Fanuc TP program (LS listing): WALL.LS

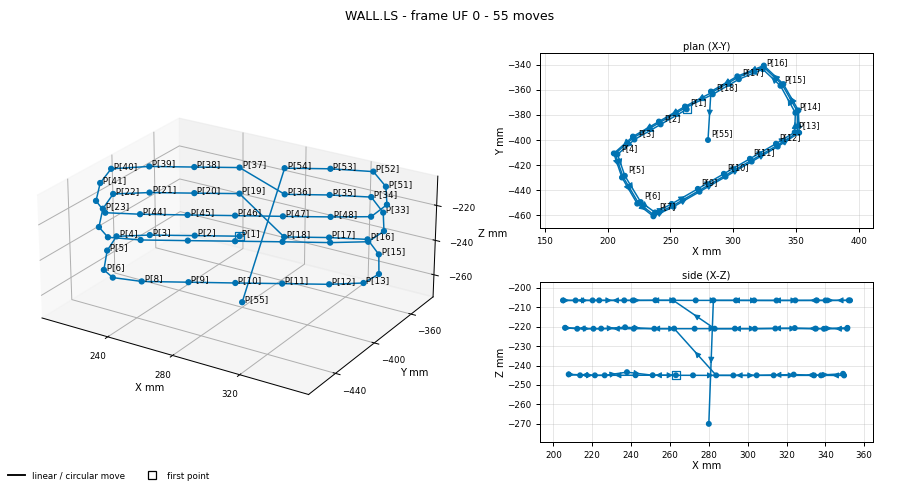
[picture p0: tool path of WALL.LS in frame UF 0, 55 of 55 moves have a stored position in this frame; points joined in program order, loops and branches not executed]
/PROG  WALL.LS
/ATTR
OWNER       = MNEDITOR;
COMMENT     = "";
PROG_SIZE   = 636;
CREATE      = DATE 23-01-07  TIME 11:59:14;
MODIFIED    = DATE 23-01-07  TIME 12:02:18;
FILE_NAME   = ;
VERSION     = 0;
LINE_COUNT  = 4;
MEMORY_SIZE = 992;
PROTECT     = READ_WRITE;
TCD:  STACK_SIZE	= 0,
      TASK_PRIORITY	= 50,
      TIME_SLICE	= 0,
      BUSY_LAMP_OFF	= 0,
      ABORT_REQUEST	= 0,
      PAUSE_REQUEST	= 0;
DEFAULT_GROUP	= 1,*,*,*,*;
CONTROL_CODE	= 00000000 00000000;
/MN
   1:J P[1] 100% FINE    ;
   2:L P[2] 100mm/sec CNT0    ;
   3:L P[3] 100mm/sec CNT0    ;
   4:L P[4] 100mm/sec CNT0    ;
   5:L P[5] 100mm/sec CNT0    ;
   6:L P[6] 100mm/sec CNT0    ;
   7:L P[7] 100mm/sec CNT0    ;
   8:L P[8] 100mm/sec CNT0    ;
   9:L P[9] 100mm/sec CNT0    ;
   10:L P[10] 100mm/sec CNT0    ;
   11:L P[11] 100mm/sec CNT0    ;
   12:L P[12] 100mm/sec CNT0    ;
   13:L P[13] 100mm/sec CNT0    ;
   14:L P[14] 100mm/sec CNT0    ;
   15:L P[15] 100mm/sec CNT0    ;
   16:L P[16] 100mm/sec CNT0    ;
   17:L P[17] 100mm/sec CNT0    ;
   18:L P[18] 100mm/sec CNT0    ;
   19:L P[19] 100mm/sec CNT0    ;
   20:L P[20] 100mm/sec CNT0    ;
   21:L P[21] 100mm/sec CNT0    ;
   22:L P[22] 100mm/sec CNT0    ;
   23:L P[23] 100mm/sec CNT0    ;
   24:L P[24] 100mm/sec CNT0    ;
   25:L P[25] 100mm/sec CNT0    ;
   26:L P[26] 100mm/sec CNT0    ;
   27:L P[27] 100mm/sec CNT0    ;
   28:L P[28] 100mm/sec CNT0    ;
   29:L P[29] 100mm/sec CNT0    ;
   30:L P[30] 100mm/sec CNT0    ;
   31:L P[31] 100mm/sec CNT0    ;
   32:L P[32] 100mm/sec CNT0    ;
   33:L P[33] 100mm/sec CNT0    ;
   34:L P[34] 100mm/sec CNT0    ;
   35:L P[35] 100mm/sec CNT0    ;
   36:L P[36] 100mm/sec CNT0    ;
   37:L P[37] 100mm/sec CNT0    ;
   38:L P[38] 100mm/sec CNT0    ;
   39:L P[39] 100mm/sec CNT0    ;
   40:L P[40] 100mm/sec CNT0    ;
   41:L P[41] 100mm/sec CNT0    ;
   42:L P[42] 100mm/sec CNT0    ;
   43:L P[43] 100mm/sec CNT0    ;
   44:L P[44] 100mm/sec CNT0    ;
   45:L P[45] 100mm/sec CNT0    ;
   46:L P[46] 100mm/sec CNT0    ;
   47:L P[47] 100mm/sec CNT0    ;
   48:L P[48] 100mm/sec CNT0    ;
   49:L P[49] 100mm/sec CNT0    ;
   50:L P[50] 100mm/sec CNT0    ;
   51:L P[51] 100mm/sec CNT0    ;
   52:L P[52] 100mm/sec CNT0    ;
   53:L P[53] 100mm/sec CNT0    ;
   54:L P[54] 100mm/sec CNT0    ;
   55:L P[55] 100mm/sec CNT0    ;
/POS
P[1]{
   GP1:
	UF : 0, UT : 6,		CONFIG : 'N U T, 0, 0, 0',
	X =  263.064  mm,	Y =   -375.561  mm,	Z =   -244.966  mm,
	W =  90.000 deg,	P =   0.000 deg,	R =   90.000 deg
};
P[2]{
   GP1:
	UF : 0, UT : 6,		CONFIG : 'N U T, 0, 0, 0',
	X =  242.275  mm,	Y =   -387.566  mm,	Z =   -244.990  mm,
	W =  90.000 deg,	P =   0.000 deg,	R =   90.000 deg
};
P[3]{
   GP1:
	UF : 0, UT : 6,		CONFIG : 'N U T, 0, 0, 0',
	X =  221.367  mm,	Y =   -399.643  mm,	Z =   -245.032  mm,
	W =  90.000 deg,	P =   0.000 deg,	R =   90.000 deg
};
P[4]{
   GP1:
	UF : 0, UT : 6,		CONFIG : 'N U T, 0, 0, 0',
	X =  207.874  mm,	Y =   -411.456  mm,	Z =   -244.528  mm,
	W =  90.000 deg,	P =   0.000 deg,	R =   90.000 deg
};
P[5]{
   GP1:
	UF : 0, UT : 6,		CONFIG : 'N U T, 0, 0, 0',
	X =  213.737  mm,	Y =   -428.487  mm,	Z =   -245.003  mm,
	W =  90.000 deg,	P =   0.000 deg,	R =   90.000 deg
};
P[6]{
   GP1:
	UF : 0, UT : 6,		CONFIG : 'N U T, 0, 0, 0',
	X =  226.401  mm,	Y =   -449.442  mm,	Z =   -245.036  mm,
	W =  90.000 deg,	P =   0.000 deg,	R =   90.000 deg
};
P[7]{
   GP1:
	UF : 0, UT : 6,		CONFIG : 'N U T, 0, 0, 0',
	X =  237.864  mm,	Y =   -457.694  mm,	Z =   -243.394  mm,
	W =  90.000 deg,	P =   0.000 deg,	R =   90.000 deg
};
P[8]{
   GP1:
	UF : 0, UT : 6,		CONFIG : 'N U T, 0, 0, 0',
	X =  251.098  mm,	Y =   -450.903  mm,	Z =   -244.977  mm,
	W =  90.000 deg,	P =   0.000 deg,	R =   90.000 deg
};
P[9]{
   GP1:
	UF : 0, UT : 6,		CONFIG : 'N U T, 0, 0, 0',
	X =  271.875  mm,	Y =   -438.904  mm,	Z =   -245.024  mm,
	W =  90.000 deg,	P =   0.000 deg,	R =   90.000 deg
};
P[10]{
   GP1:
	UF : 0, UT : 6,		CONFIG : 'N U T, 0, 0, 0',
	X =  292.641  mm,	Y =   -426.910  mm,	Z =   -245.078  mm,
	W =  90.000 deg,	P =   0.000 deg,	R =   90.000 deg
};
P[11]{
   GP1:
	UF : 0, UT : 6,		CONFIG : 'N U T, 0, 0, 0',
	X =  313.392  mm,	Y =   -414.931  mm,	Z =   -245.046  mm,
	W =  90.000 deg,	P =   0.000 deg,	R =   90.000 deg
};
P[12]{
   GP1:
	UF : 0, UT : 6,		CONFIG : 'N U T, 0, 0, 0',
	X =  334.179  mm,	Y =   -402.928  mm,	Z =   -245.053  mm,
	W =  90.000 deg,	P =   0.000 deg,	R =   90.000 deg
};
P[13]{
   GP1:
	UF : 0, UT : 6,		CONFIG : 'N U T, 0, 0, 0',
	X =  349.100  mm,	Y =   -393.829  mm,	Z =   -244.223  mm,
	W =  90.000 deg,	P =   0.000 deg,	R =   90.000 deg
};
P[14]{
   GP1:
	UF : 0, UT : 6,		CONFIG : 'N U T, 0, 0, 0',
	X =  349.628  mm,	Y =   -378.344  mm,	Z =   -245.091  mm,
	W =  90.000 deg,	P =   0.000 deg,	R =   90.000 deg
};
P[15]{
   GP1:
	UF : 0, UT : 6,		CONFIG : 'N U T, 0, 0, 0',
	X =  337.749  mm,	Y =   -356.772  mm,	Z =   -245.043  mm,
	W =  90.000 deg,	P =   0.000 deg,	R =   90.000 deg
};
P[16]{
   GP1:
	UF : 0, UT : 6,		CONFIG : 'N U T, 0, 0, 0',
	X =  323.686  mm,	Y =   -343.563  mm,	Z =   -244.638  mm,
	W =  90.000 deg,	P =   0.000 deg,	R =   90.000 deg
};
P[17]{
   GP1:
	UF : 0, UT : 6,		CONFIG : 'N U T, 0, 0, 0',
	X =  304.635  mm,	Y =   -351.562  mm,	Z =   -245.020  mm,
	W =  90.000 deg,	P =   0.000 deg,	R =   90.000 deg
};
P[18]{
   GP1:
	UF : 0, UT : 6,		CONFIG : 'N U T, 0, 0, 0',
	X =  283.803  mm,	Y =   -363.591  mm,	Z =   -245.029  mm,
	W =  90.000 deg,	P =   0.000 deg,	R =   90.000 deg
};
P[19]{
   GP1:
	UF : 0, UT : 6,		CONFIG : 'N U T, 0, 0, 0',
	X =  262.167  mm,	Y =   -374.140  mm,	Z =   -220.957  mm,
	W =  90.000 deg,	P =   0.000 deg,	R =   90.000 deg
};
P[20]{
   GP1:
	UF : 0, UT : 6,		CONFIG : 'N U T, 0, 0, 0',
	X =  241.342  mm,	Y =   -386.170  mm,	Z =   -221.026  mm,
	W =  90.000 deg,	P =   0.000 deg,	R =   90.000 deg
};
P[21]{
   GP1:
	UF : 0, UT : 6,		CONFIG : 'N U T, 0, 0, 0',
	X =  220.631  mm,	Y =   -398.129  mm,	Z =   -221.039  mm,
	W =  90.000 deg,	P =   0.000 deg,	R =   90.000 deg
};
P[22]{
   GP1:
	UF : 0, UT : 6,		CONFIG : 'N U T, 0, 0, 0',
	X =  205.989  mm,	Y =   -410.913  mm,	Z =   -220.558  mm,
	W =  90.000 deg,	P =   0.000 deg,	R =   90.000 deg
};
P[23]{
   GP1:
	UF : 0, UT : 6,		CONFIG : 'N U T, 0, 0, 0',
	X =  212.279  mm,	Y =   -429.315  mm,	Z =   -221.051  mm,
	W =  90.000 deg,	P =   0.000 deg,	R =   90.000 deg
};
P[24]{
   GP1:
	UF : 0, UT : 6,		CONFIG : 'N U T, 0, 0, 0',
	X =  224.597  mm,	Y =   -450.243  mm,	Z =   -220.970  mm,
	W =  90.000 deg,	P =   0.000 deg,	R =   90.000 deg
};
P[25]{
   GP1:
	UF : 0, UT : 6,		CONFIG : 'N U T, 0, 0, 0',
	X =  236.910  mm,	Y =   -459.701  mm,	Z =   -220.287  mm,
	W =  90.000 deg,	P =   0.000 deg,	R =   90.000 deg
};
P[26]{
   GP1:
	UF : 0, UT : 6,		CONFIG : 'N U T, 0, 0, 0',
	X =  251.946  mm,	Y =   -452.348  mm,	Z =   -221.034  mm,
	W =  90.000 deg,	P =   0.000 deg,	R =   90.000 deg
};
P[27]{
   GP1:
	UF : 0, UT : 6,		CONFIG : 'N U T, 0, 0, 0',
	X =  272.697  mm,	Y =   -440.367  mm,	Z =   -221.028  mm,
	W =  90.000 deg,	P =   0.000 deg,	R =   90.000 deg
};
P[28]{
   GP1:
	UF : 0, UT : 6,		CONFIG : 'N U T, 0, 0, 0',
	X =  293.446  mm,	Y =   -428.391  mm,	Z =   -220.980  mm,
	W =  90.000 deg,	P =   0.000 deg,	R =   90.000 deg
};
P[29]{
   GP1:
	UF : 0, UT : 6,		CONFIG : 'N U T, 0, 0, 0',
	X =  314.251  mm,	Y =   -416.382  mm,	Z =   -220.936  mm,
	W =  90.000 deg,	P =   0.000 deg,	R =   90.000 deg
};
P[30]{
   GP1:
	UF : 0, UT : 6,		CONFIG : 'N U T, 0, 0, 0',
	X =  335.102  mm,	Y =   -404.336  mm,	Z =   -221.012  mm,
	W =  90.000 deg,	P =   0.000 deg,	R =   90.000 deg
};
P[31]{
   GP1:
	UF : 0, UT : 6,		CONFIG : 'N U T, 0, 0, 0',
	X =  351.351  mm,	Y =   -394.060  mm,	Z =   -220.582  mm,
	W =  90.000 deg,	P =   0.000 deg,	R =   90.000 deg
};
P[32]{
   GP1:
	UF : 0, UT : 6,		CONFIG : 'N U T, 0, 0, 0',
	X =  351.165  mm,	Y =   -377.074  mm,	Z =   -221.045  mm,
	W =  90.000 deg,	P =   0.000 deg,	R =   90.000 deg
};
P[33]{
   GP1:
	UF : 0, UT : 6,		CONFIG : 'N U T, 0, 0, 0',
	X =  339.240  mm,	Y =   -356.000  mm,	Z =   -221.074  mm,
	W =  90.000 deg,	P =   0.000 deg,	R =   90.000 deg
};
P[34]{
   GP1:
	UF : 0, UT : 6,		CONFIG : 'N U T, 0, 0, 0',
	X =  324.236  mm,	Y =   -341.710  mm,	Z =   -220.699  mm,
	W =  90.000 deg,	P =   0.000 deg,	R =   90.000 deg
};
P[35]{
   GP1:
	UF : 0, UT : 6,		CONFIG : 'N U T, 0, 0, 0',
	X =  303.694  mm,	Y =   -350.169  mm,	Z =   -221.036  mm,
	W =  90.000 deg,	P =   0.000 deg,	R =   90.000 deg
};
P[36]{
   GP1:
	UF : 0, UT : 6,		CONFIG : 'N U T, 0, 0, 0',
	X =  283.011  mm,	Y =   -362.109  mm,	Z =   -221.014  mm,
	W =  90.000 deg,	P =   0.000 deg,	R =   90.000 deg
};
P[37]{
   GP1:
	UF : 0, UT : 6,		CONFIG : 'N U T, 0, 0, 0',
	X =  261.677  mm,	Y =   -373.250  mm,	Z =   -206.429  mm,
	W =  90.000 deg,	P =   0.000 deg,	R =   90.000 deg
};
P[38]{
   GP1:
	UF : 0, UT : 6,		CONFIG : 'N U T, 0, 0, 0',
	X =  240.881  mm,	Y =   -385.261  mm,	Z =   -206.472  mm,
	W =  90.000 deg,	P =   0.000 deg,	R =   90.000 deg
};
P[39]{
   GP1:
	UF : 0, UT : 6,		CONFIG : 'N U T, 0, 0, 0',
	X =  220.167  mm,	Y =   -397.220  mm,	Z =   -206.458  mm,
	W =  90.000 deg,	P =   0.000 deg,	R =   90.000 deg
};
P[40]{
   GP1:
	UF : 0, UT : 6,		CONFIG : 'N U T, 0, 0, 0',
	X =  204.931  mm,	Y =   -410.680  mm,	Z =   -206.454  mm,
	W =  90.000 deg,	P =   0.000 deg,	R =   90.000 deg
};
P[41]{
   GP1:
	UF : 0, UT : 6,		CONFIG : 'N U T, 0, 0, 0',
	X =  211.430  mm,	Y =   -429.882  mm,	Z =   -206.475  mm,
	W =  90.000 deg,	P =   0.000 deg,	R =   90.000 deg
};
P[42]{
   GP1:
	UF : 0, UT : 6,		CONFIG : 'N U T, 0, 0, 0',
	X =  223.588  mm,	Y =   -450.719  mm,	Z =   -206.440  mm,
	W =  90.000 deg,	P =   0.000 deg,	R =   90.000 deg
};
P[43]{
   GP1:
	UF : 0, UT : 6,		CONFIG : 'N U T, 0, 0, 0',
	X =  236.477  mm,	Y =   -460.831  mm,	Z =   -206.445  mm,
	W =  90.000 deg,	P =   0.000 deg,	R =   90.000 deg
};
P[44]{
   GP1:
	UF : 0, UT : 6,		CONFIG : 'N U T, 0, 0, 0',
	X =  252.504  mm,	Y =   -453.208  mm,	Z =   -206.401  mm,
	W =  90.000 deg,	P =   0.000 deg,	R =   90.000 deg
};
P[45]{
   GP1:
	UF : 0, UT : 6,		CONFIG : 'N U T, 0, 0, 0',
	X =  273.258  mm,	Y =   -441.221  mm,	Z =   -206.450  mm,
	W =  90.000 deg,	P =   0.000 deg,	R =   90.000 deg
};
P[46]{
   GP1:
	UF : 0, UT : 6,		CONFIG : 'N U T, 0, 0, 0',
	X =  293.998  mm,	Y =   -429.245  mm,	Z =   -206.452  mm,
	W =  90.000 deg,	P =   0.000 deg,	R =   90.000 deg
};
P[47]{
   GP1:
	UF : 0, UT : 6,		CONFIG : 'N U T, 0, 0, 0',
	X =  314.843  mm,	Y =   -417.205  mm,	Z =   -206.504  mm,
	W =  90.000 deg,	P =   0.000 deg,	R =   90.000 deg
};
P[48]{
   GP1:
	UF : 0, UT : 6,		CONFIG : 'N U T, 0, 0, 0',
	X =  335.587  mm,	Y =   -405.232  mm,	Z =   -206.449  mm,
	W =  90.000 deg,	P =   0.000 deg,	R =   90.000 deg
};
P[49]{
   GP1:
	UF : 0, UT : 6,		CONFIG : 'N U T, 0, 0, 0',
	X =  352.687  mm,	Y =   -394.191  mm,	Z =   -206.456  mm,
	W =  90.000 deg,	P =   0.000 deg,	R =   90.000 deg
};
P[50]{
   GP1:
	UF : 0, UT : 6,		CONFIG : 'N U T, 0, 0, 0',
	X =  352.066  mm,	Y =   -376.389  mm,	Z =   -206.425  mm,
	W =  90.000 deg,	P =   0.000 deg,	R =   90.000 deg
};
P[51]{
   GP1:
	UF : 0, UT : 6,		CONFIG : 'N U T, 0, 0, 0',
	X =  340.074  mm,	Y =   -355.402  mm,	Z =   -206.467  mm,
	W =  90.000 deg,	P =   0.000 deg,	R =   90.000 deg
};
P[52]{
   GP1:
	UF : 0, UT : 6,		CONFIG : 'N U T, 0, 0, 0',
	X =  324.525  mm,	Y =   -340.629  mm,	Z =   -206.457  mm,
	W =  90.000 deg,	P =   0.000 deg,	R =   90.000 deg
};
P[53]{
   GP1:
	UF : 0, UT : 6,		CONFIG : 'N U T, 0, 0, 0',
	X =  303.339  mm,	Y =   -349.197  mm,	Z =   -206.453  mm,
	W =  90.000 deg,	P =   0.000 deg,	R =   90.000 deg
};
P[54]{
   GP1:
	UF : 0, UT : 6,		CONFIG : 'N U T, 0, 0, 0',
	X =  282.347  mm,	Y =   -361.317  mm,	Z =   -206.444  mm,
	W =  90.000 deg,	P =   0.000 deg,	R =   90.000 deg
};
P[55]{
   GP1:
	UF : 0, UT : 6,		CONFIG : 'N U T, 0, 0, 0',
	X =  280.000  mm,	Y =   -400.000  mm,	Z =   -270.000  mm,
	W =  90.000 deg,	P =   0.000 deg,	R =   90.000 deg
};
/END
